(* CODESYS project TRIFASICO.project

Project tree, tasks and I/O mapping:
  Device : CODESYS Control Win V3, 3S - Smart Software Solutions GmbH, order no. 305021, version 3.5.11.30
    application Application
      libraries: Standard, * (System)
      task MainTask (cyclic, interval t#20ms, priority 1) calls PLC_PRG
      program PLC_PRG [LD]
*)

// Device/Application/PLC_PRG
PROGRAM PLC_PRG
VAR
	S1 : BOOL;           // BOTAO DE PARTIDA
	K1A : BOOL;          // MERKER DE RELE AUXILIAR
	K2A : BOOL;          // ERKER DE RELE AUXILIAR
	S2 : BOOL;           // BOTAODE PARADA
	KT1 : BOOL;         // TEMPORIZADOR TRABALHO
	KT2 : BOOL;         // TEMPORIZADOR PAUSA
	KM1 : BOOL;         // CONTATOR MOTOR
	H1 : BOOL;          // LAMPADA MOTOR
	FR : BOOL;          // TERMICA
END_VAR

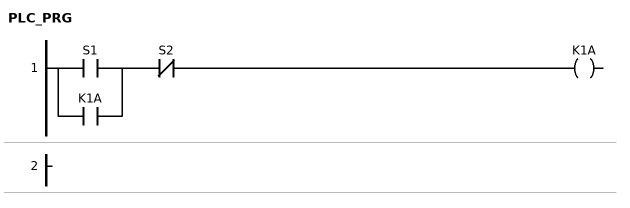
// NETWORK 1
K1A := (S1 OR K1A) AND NOT S2;

// NETWORK 2

END_PROGRAM
